{attribute 'qualified_only'}
{attribute 'strict'}
TYPE E_LAMP_RPC_ERROR :
(
	OK						:= 0,
	NOT_OP					:= -1,			
	NOT_NOTOP_READY			:= -2,			
	NOT_NOTOP_NOTREADY		:= -3,			
	SWITCHING_ON			:= -4,			
	SWITCHING_OFF			:= -5,			
	COOLING					:= -6,			
	LOCAL					:= -7			
);
END_TYPE

(* stored: Version 1.1.0.1, ProductVersion 3.1.4022.16
   DUT E_LAMP_RPC_ERROR: Id {ae0abd72-7773-43bc-83e5-11d973ea74e5} *)
